// TIA Portal V17 export
// export: Created 2023-12-22T15:05:34.5254244Z, ExportSetting WithDefaults, DisplayName Totally Integrated Automation Portal, DisplayVersion V17, DisplayName TIA Portal Openness, DisplayVersion V17, DisplayName TIA Portal Version Control Interface, DisplayVersion V17, DisplayName STEP 7 Professional, DisplayVersion V17, DisplayName STEP 7 Safety, DisplayVersion V17, DisplayName WinCC Advanced, DisplayVersion V17
DATA_BLOCK "Smena_DB"   // DB26
VERSION : 0.1
// stored: AutoNumber true, DBAccessibleFromOPCUA true, InstanceOfName Smena, InstanceOfType FB
"Smena"
   // VAR RETAIN
   //    ON_1 : Struct
   //       Use : Bool := FALSE;
   //       H : Int := 10;
   //       "M" : Int := 12;
   //    END_STRUCT;
   //    ON_2 : Struct
   //       Use : Bool := FALSE;
   //       H : Int := 10;
   //       "M" : Int := 9;
   //    END_STRUCT;
   //    pos : Array[0..31] of Bool;
   //    Line_1 : Array[0..2] of Struct
   //       Water : Real;
   //       Reagent : Real;
   //    END_STRUCT;
   //    Line_2 : Array[0..2] of Struct
   //       Water : Real;
   //       Reagent : Real;
   //    END_STRUCT;
   //    "Time" : Array[0..2] of Struct
   //       Start_H : Int;
   //       Start_M : Int;
   //       "Date" : Int;
   //       Mounth : Int;
   //    END_STRUCT;
   //    Time_DTL : DTL := DTL#2020-10-19-10:13:30.152898937;
   // END_VAR
BEGIN
   pos[0..31] := FALSE;
   Line_1[0..2].Water := 0.0;
   Line_1[0..2].Reagent := 0.0;
   Line_2[0..2].Water := 0.0;
   Line_2[0..2].Reagent := 0.0;
   "Time"[0].Start_H := 0;
   "Time"[1].Start_H := 10;
   "Time"[2].Start_H := 6;
   "Time"[0].Start_M := 0;
   "Time"[1].Start_M := 9;
   "Time"[2].Start_M := 0;
   "Time"[0]."Date" := 0;
   "Time"[1..2]."Date" := 10;
   "Time"[0].Mounth := 0;
   "Time"[1].Mounth := 12;
   "Time"[2].Mounth := 9;
END_DATA_BLOCK
